VAR_GLOBAL
	
	(*****P07_CapPusher********)	  
	IbCapPusher0DoorsOpen 				AT %I* :BOOL;
	//Szlaban
	bCapPusherManualGate						:BOOL;						// Szlaban formatki		
	
	//Podajnik 
	iCapPusherFeederState						:INT;						// Stan
	sCapPusherFeederState						:STRING;					// Stan
    bCapPusherFeederHoming						:BOOL;						// Bazowanie
 	bCapPusherFeederRun							:BOOL; 						// Cykl
	bCapPusherFeederIgnoreErrors				:BOOL;					 	// Ignoruj błędy
	bCapPusherFeederHeightSet					:BOOL;						// Ustaw
	bCapPusherFeederManualSorterEngine			:BOOL;						// Silnik
	bCapPusherFeederManualSorterVibrator		:BOOL;						// Wibrator
	bCapPusherFeederManualSorterVibrator2		:BOOL;						// Wibrator
	bCapPusherFeederManualSorterAir				:BOOL;						// Wydmuch

	//Zakrecanie
	iCapPusherState								:INT;						// Stan
	sCapPusherState								:STRING;					// Stan
    bCapPusherHoming							:BOOL;						// Bazowanie
 	bCapPusherRun								:BOOL; 						// Cykl
	bCapPusherIgnoreErrors						:BOOL;					 	// Ignoruj błędy
	bCapPusherHeightSet							:BOOL;						// Ustaw
	bCapPusherManualPusher						:BOOL;						// Wbijak
	bCapPusherManualBlockActuator				:BOOL;						// Boczny	
	bCapPusherManualFormPositioning				:BOOL;						// Pozycjonowanie formatek
	
	(*****P00_Recipes*******)	  
	//Szlaban

	//Podajnik                     				
	iCapPusherFeederTimeDelayOnShow				:INT; 						// Opóźnienie włączenia
	iCapPusherFeederTimeDelayOffShow			:INT; 						// Opóźnienie wyłączenia
	iCapPusherFeederTimeToEmptySleeveErrorShow	:INT;						// Czas do alarmu pustego rękawa [s] (10-120 s)

	//Zakrecanie                    				
	bCapPusherEnableShow						:BOOL;						// Aktywacja
	iCapPusherTimeShow							:INT; 						// Czas wibjania
	iCapPusherTime2Show							:INT;						// Czas 2

END_VAR

(* stored: Version 1.2.0.0, ProductVersion 3.1.4026.13, FileIdentifier 230f3303ab0d6eba2fe06ab8b37339ac0d0273d8, FileSignature 1b3d1e5e717165022140df3b7a10d7e34fc1676a18a635401a90dc3613fcb67291811b4a81e02b7aaa8044657b278668d7e493365f2e73f705a5bdcc046e1fbc4ee1bd07df9d661170196dbba98455357ae9d7820308e69b8c58116de8613a0f9d1c4ef9bee1bb6f5a7c72c9b6c8d1e4038caf51e5e43aeab7ec21435c75140891adea8d9a2c2fb9d6476a12e013ba9451bc488eef90df192eb8ac3ad627420484efdb5fb158ae8b2a317d5a43e42fdacad52a8c4fd8715bf542fcc9626e1d2894de268042b40318834d9961268acfa50be833867be40f4031dcbddfca4c390390554493592c70533a87e802e607c3beff2101b6a4911bc92b19d26a8021641a
   GVL VIS_CP: Id {a3713359-d7e5-496c-a5b4-e777826a4d25} *)
